ABB RAPID module: 9b54fd59.mod

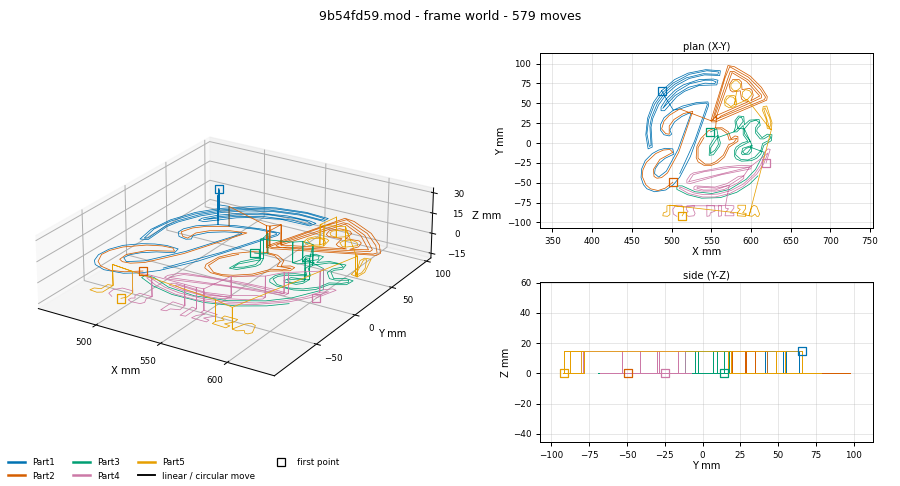
[picture p0: tool path of 9b54fd59.mod in frame world, 579 of 581 moves have a stored position in this frame; points joined in program order, loops and branches not executed]
MODULE ImageDraw
  ! Generated 2026-10-06 12:25 for ABB GoFa CRB 15000: 38 strokes
  PERS tooldata tPen:=[TRUE,[[0,0,120.0],[1,0,0,0]],[0.3,[0,0,60.0],[1,0,0,0],0,0,0]];
  PERS wobjdata wPaper:=[FALSE,TRUE,"",[[400,-110,0],[1,0,0,0]],[[0,0,0],[1,0,0,0]]];
  CONST robtarget pOrigin:=[[0,0,0],[0,1,0,0],[0,0,0,0],[9E9,9E9,9E9,9E9,9E9,9E9]];
  CONST jointtarget jHome:=[[0,0,0,0,30,0],[9E9,9E9,9E9,9E9,9E9,9E9]];
  CONST speeddata vDraw:=[40,100,5000,1000];
  CONST speeddata vApproach:=[20,100,5000,1000];
  CONST speeddata vTravel:=[200,200,5000,1000];

  PROC DrawImage()
    ConfL\Off;
    ConfJ\Off;
    MoveAbsJ jHome\NoEOffs,vTravel,fine,tPen;
    Part1;
    Part2;
    Part3;
    Part4;
    Part5;
    MoveAbsJ jHome\NoEOffs,vTravel,fine,tPen;
  ENDPROC

  PROC Part1()
    MoveL Offs(pOrigin,87.5,175.8,15.0),vTravel,z5,tPen\WObj:=wPaper;
    MoveL Offs(pOrigin,87.5,175.8,0.0),vApproach,fine,tPen\WObj:=wPaper;
    MoveL Offs(pOrigin,77.2,161.0,0.0),vDraw,z1,tPen\WObj:=wPaper;
    MoveL Offs(pOrigin,69.8,141.1,0.0),vDraw,z1,tPen\WObj:=wPaper;
    MoveL Offs(pOrigin,67.6,120.4,0.0),vDraw,z1,tPen\WObj:=wPaper;
    MoveL Offs(pOrigin,70.5,102.6,0.0),vDraw,z1,tPen\WObj:=wPaper;
    MoveL Offs(pOrigin,75.7,104.8,0.0),vDraw,z1,tPen\WObj:=wPaper;
    MoveL Offs(pOrigin,74.2,130.0,0.0),vDraw,z1,tPen\WObj:=wPaper;
    MoveL Offs(pOrigin,76.4,141.1,0.0),vDraw,z1,tPen\WObj:=wPaper;
    MoveL Offs(pOrigin,83.8,158.1,0.0),vDraw,z1,tPen\WObj:=wPaper;
    MoveL Offs(pOrigin,93.4,171.4,0.0),vDraw,z1,tPen\WObj:=wPaper;
    MoveL Offs(pOrigin,106.0,182.5,0.0),vDraw,z1,tPen\WObj:=wPaper;
    MoveL Offs(pOrigin,122.3,191.3,0.0),vDraw,z1,tPen\WObj:=wPaper;
    MoveL Offs(pOrigin,141.5,195.8,0.0),vDraw,z1,tPen\WObj:=wPaper;
    MoveL Offs(pOrigin,160.7,195.0,0.0),vDraw,z1,tPen\WObj:=wPaper;
    MoveL Offs(pOrigin,161.5,201.0,0.0),vDraw,z1,tPen\WObj:=wPaper;
    MoveL Offs(pOrigin,143.0,202.4,0.0),vDraw,z1,tPen\WObj:=wPaper;
    MoveL Offs(pOrigin,120.8,198.0,0.0),vDraw,z1,tPen\WObj:=wPaper;
    MoveL Offs(pOrigin,103.8,189.9,0.0),vDraw,z1,tPen\WObj:=wPaper;
    MoveL Offs(pOrigin,87.5,175.8,0.0),vDraw,fine,tPen\WObj:=wPaper;
    MoveL Offs(pOrigin,87.5,175.8,15.0),vApproach,z5,tPen\WObj:=wPaper;
    MoveL Offs(pOrigin,89.0,173.6,15.0),vTravel,z5,tPen\WObj:=wPaper;
    MoveL Offs(pOrigin,89.0,173.6,0.0),vApproach,fine,tPen\WObj:=wPaper;
    MoveL Offs(pOrigin,101.6,185.4,0.0),vDraw,z1,tPen\WObj:=wPaper;
    MoveL Offs(pOrigin,122.3,196.5,0.0),vDraw,z1,tPen\WObj:=wPaper;
    MoveL Offs(pOrigin,144.5,201.0,0.0),vDraw,z1,tPen\WObj:=wPaper;
    MoveL Offs(pOrigin,159.2,199.5,0.0),vDraw,z1,tPen\WObj:=wPaper;
    MoveL Offs(pOrigin,158.5,196.5,0.0),vDraw,z1,tPen\WObj:=wPaper;
    MoveL Offs(pOrigin,140.0,197.3,0.0),vDraw,z1,tPen\WObj:=wPaper;
    MoveL Offs(pOrigin,118.6,192.1,0.0),vDraw,z1,tPen\WObj:=wPaper;
    MoveL Offs(pOrigin,103.8,183.9,0.0),vDraw,z1,tPen\WObj:=wPaper;
    MoveL Offs(pOrigin,92.7,174.3,0.0),vDraw,z1,tPen\WObj:=wPaper;
    MoveL Offs(pOrigin,82.3,160.3,0.0),vDraw,z1,tPen\WObj:=wPaper;
    MoveL Offs(pOrigin,74.9,142.5,0.0),vDraw,z1,tPen\WObj:=wPaper;
    MoveL Offs(pOrigin,72.7,131.4,0.0),vDraw,z1,tPen\WObj:=wPaper;
    MoveL Offs(pOrigin,74.2,107.0,0.0),vDraw,z1,tPen\WObj:=wPaper;
    MoveL Offs(pOrigin,72.0,105.6,0.0),vDraw,z1,tPen\WObj:=wPaper;
    MoveL Offs(pOrigin,69.0,121.8,0.0),vDraw,z1,tPen\WObj:=wPaper;
    MoveL Offs(pOrigin,71.2,139.6,0.0),vDraw,z1,tPen\WObj:=wPaper;
    MoveL Offs(pOrigin,78.6,158.8,0.0),vDraw,z1,tPen\WObj:=wPaper;
    MoveL Offs(pOrigin,89.0,173.6,0.0),vDraw,fine,tPen\WObj:=wPaper;
    MoveL Offs(pOrigin,89.0,173.6,15.0),vApproach,z5,tPen\WObj:=wPaper;
    MoveL Offs(pOrigin,93.4,165.5,15.0),vTravel,z5,tPen\WObj:=wPaper;
    MoveL Offs(pOrigin,93.4,165.5,0.0),vApproach,fine,tPen\WObj:=wPaper;
    MoveL Offs(pOrigin,86.8,155.1,0.0),vDraw,z1,tPen\WObj:=wPaper;
    MoveL Offs(pOrigin,86.8,150.7,0.0),vDraw,z1,tPen\WObj:=wPaper;
    MoveL Offs(pOrigin,91.2,150.7,0.0),vDraw,z1,tPen\WObj:=wPaper;
    MoveL Offs(pOrigin,106.7,168.4,0.0),vDraw,z1,tPen\WObj:=wPaper;
    MoveL Offs(pOrigin,116.4,175.1,0.0),vDraw,z1,tPen\WObj:=wPaper;
    MoveL Offs(pOrigin,134.8,182.5,0.0),vDraw,z1,tPen\WObj:=wPaper;
    MoveL Offs(pOrigin,157.0,183.2,0.0),vDraw,z1,tPen\WObj:=wPaper;
    MoveL Offs(pOrigin,158.5,189.1,0.0),vDraw,z1,tPen\WObj:=wPaper;
    MoveL Offs(pOrigin,152.6,190.6,0.0),vDraw,z1,tPen\WObj:=wPaper;
    MoveL Offs(pOrigin,134.8,189.9,0.0),vDraw,z1,tPen\WObj:=wPaper;
    MoveL Offs(pOrigin,114.9,183.2,0.0),vDraw,z1,tPen\WObj:=wPaper;
    MoveL Offs(pOrigin,104.5,176.5,0.0),vDraw,z1,tPen\WObj:=wPaper;
    MoveL Offs(pOrigin,93.4,165.5,0.0),vDraw,fine,tPen\WObj:=wPaper;
    MoveL Offs(pOrigin,93.4,165.5,15.0),vApproach,z5,tPen\WObj:=wPaper;
    MoveL Offs(pOrigin,94.9,163.2,15.0),vTravel,z5,tPen\WObj:=wPaper;
    MoveL Offs(pOrigin,94.9,163.2,0.0),vApproach,fine,tPen\WObj:=wPaper;
    MoveL Offs(pOrigin,106.7,175.1,0.0),vDraw,z1,tPen\WObj:=wPaper;
    MoveL Offs(pOrigin,123.0,184.7,0.0),vDraw,z1,tPen\WObj:=wPaper;
    MoveL Offs(pOrigin,142.2,189.1,0.0),vDraw,z1,tPen\WObj:=wPaper;
    MoveL Offs(pOrigin,151.1,189.1,0.0),vDraw,z1,tPen\WObj:=wPaper;
    MoveL Offs(pOrigin,156.3,186.9,0.0),vDraw,z1,tPen\WObj:=wPaper;
    MoveL Offs(pOrigin,154.1,184.7,0.0),vDraw,z1,tPen\WObj:=wPaper;
    MoveL Offs(pOrigin,142.2,185.4,0.0),vDraw,z1,tPen\WObj:=wPaper;
    MoveL Offs(pOrigin,121.5,180.2,0.0),vDraw,z1,tPen\WObj:=wPaper;
    MoveL Offs(pOrigin,104.5,169.9,0.0),vDraw,z1,tPen\WObj:=wPaper;
    MoveL Offs(pOrigin,89.0,153.6,0.0),vDraw,z1,tPen\WObj:=wPaper;
    MoveL Offs(pOrigin,94.9,163.2,0.0),vDraw,fine,tPen\WObj:=wPaper;
    MoveL Offs(pOrigin,94.9,163.2,15.0),vApproach,z5,tPen\WObj:=wPaper;
    MoveL Offs(pOrigin,102.3,151.4,15.0),vTravel,z5,tPen\WObj:=wPaper;
    MoveL Offs(pOrigin,102.3,151.4,0.0),vApproach,fine,tPen\WObj:=wPaper;
    MoveL Offs(pOrigin,90.5,141.8,0.0),vDraw,z1,tPen\WObj:=wPaper;
    MoveL Offs(pOrigin,86.0,132.9,0.0),vDraw,z1,tPen\WObj:=wPaper;
    MoveL Offs(pOrigin,86.0,126.3,0.0),vDraw,z1,tPen\WObj:=wPaper;
    MoveL Offs(pOrigin,90.5,120.4,0.0),vDraw,z1,tPen\WObj:=wPaper;
    MoveL Offs(pOrigin,97.1,118.9,0.0),vDraw,z1,tPen\WObj:=wPaper;
    MoveL Offs(pOrigin,100.1,121.1,0.0),vDraw,z1,tPen\WObj:=wPaper;
    MoveL Offs(pOrigin,97.9,126.3,0.0),vDraw,z1,tPen\WObj:=wPaper;
    MoveL Offs(pOrigin,103.8,136.6,0.0),vDraw,z1,tPen\WObj:=wPaper;
    MoveL Offs(pOrigin,112.7,143.3,0.0),vDraw,z1,tPen\WObj:=wPaper;
    MoveL Offs(pOrigin,122.3,147.7,0.0),vDraw,z1,tPen\WObj:=wPaper;
    MoveL Offs(pOrigin,124.5,147.0,0.0),vDraw,z1,tPen\WObj:=wPaper;
    MoveL Offs(pOrigin,108.2,101.9,0.0),vDraw,z1,tPen\WObj:=wPaper;
    MoveL Offs(pOrigin,93.4,74.5,0.0),vDraw,z1,tPen\WObj:=wPaper;
    MoveL Offs(pOrigin,83.8,67.1,0.0),vDraw,z1,tPen\WObj:=wPaper;
    MoveL Offs(pOrigin,78.6,71.5,0.0),vDraw,z1,tPen\WObj:=wPaper;
    MoveL Offs(pOrigin,79.4,77.5,0.0),vDraw,z1,tPen\WObj:=wPaper;
    MoveL Offs(pOrigin,83.8,84.1,0.0),vDraw,z1,tPen\WObj:=wPaper;
    MoveL Offs(pOrigin,92.0,90.8,0.0),vDraw,z1,tPen\WObj:=wPaper;
    MoveL Offs(pOrigin,103.0,96.0,0.0),vDraw,z1,tPen\WObj:=wPaper;
    MoveL Offs(pOrigin,101.6,102.6,0.0),vDraw,z1,tPen\WObj:=wPaper;
    MoveL Offs(pOrigin,92.0,103.3,0.0),vDraw,z1,tPen\WObj:=wPaper;
    MoveL Offs(pOrigin,83.8,101.1,0.0),vDraw,z1,tPen\WObj:=wPaper;
    MoveL Offs(pOrigin,75.7,96.7,0.0),vDraw,z1,tPen\WObj:=wPaper;
    MoveL Offs(pOrigin,66.8,87.8,0.0),vDraw,z1,tPen\WObj:=wPaper;
    MoveL Offs(pOrigin,62.4,77.5,0.0),vDraw,z1,tPen\WObj:=wPaper;
    MoveL Offs(pOrigin,61.6,66.4,0.0),vDraw,z1,tPen\WObj:=wPaper;
    MoveL Offs(pOrigin,64.6,57.5,0.0),vDraw,z1,tPen\WObj:=wPaper;
    MoveL Offs(pOrigin,69.0,52.3,0.0),vDraw,z1,tPen\WObj:=wPaper;
    MoveL Offs(pOrigin,78.6,48.6,0.0),vDraw,z1,tPen\WObj:=wPaper;
    MoveL Offs(pOrigin,92.7,50.8,0.0),vDraw,z1,tPen\WObj:=wPaper;
    MoveL Offs(pOrigin,102.3,57.5,0.0),vDraw,z1,tPen\WObj:=wPaper;
    MoveL Offs(pOrigin,110.4,67.1,0.0),vDraw,z1,tPen\WObj:=wPaper;
    MoveL Offs(pOrigin,123.8,93.0,0.0),vDraw,z1,tPen\WObj:=wPaper;
    MoveL Offs(pOrigin,146.7,157.3,0.0),vDraw,z1,tPen\WObj:=wPaper;
    MoveL Offs(pOrigin,145.9,161.8,0.0),vDraw,z1,tPen\WObj:=wPaper;
    MoveL Offs(pOrigin,131.9,161.0,0.0),vDraw,z1,tPen\WObj:=wPaper;
    MoveL Offs(pOrigin,114.1,156.6,0.0),vDraw,z1,tPen\WObj:=wPaper;
    MoveL Offs(pOrigin,102.3,151.4,0.0),vDraw,fine,tPen\WObj:=wPaper;
    MoveL Offs(pOrigin,102.3,151.4,15.0),vApproach,z5,tPen\WObj:=wPaper;
    MoveL Offs(pOrigin,110.4,152.9,15.0),vTravel,z5,tPen\WObj:=wPaper;
    MoveL Offs(pOrigin,110.4,152.9,0.0),vApproach,fine,tPen\WObj:=wPaper;
    MoveL Offs(pOrigin,128.9,158.8,0.0),vDraw,z1,tPen\WObj:=wPaper;
    MoveL Offs(pOrigin,143.7,160.3,0.0),vDraw,z1,tPen\WObj:=wPaper;
    MoveL Offs(pOrigin,145.2,158.8,0.0),vDraw,z1,tPen\WObj:=wPaper;
    MoveL Offs(pOrigin,128.9,112.2,0.0),vDraw,z1,tPen\WObj:=wPaper;
    MoveL Offs(pOrigin,110.4,71.5,0.0),vDraw,z1,tPen\WObj:=wPaper;
  ENDPROC

  PROC Part2()
    MoveL Offs(pOrigin,101.6,60.5,0.0),vDraw,z1,tPen\WObj:=wPaper;
    MoveL Offs(pOrigin,92.0,53.1,0.0),vDraw,z1,tPen\WObj:=wPaper;
    MoveL Offs(pOrigin,83.1,50.1,0.0),vDraw,z1,tPen\WObj:=wPaper;
    MoveL Offs(pOrigin,73.5,52.3,0.0),vDraw,z1,tPen\WObj:=wPaper;
    MoveL Offs(pOrigin,67.6,57.5,0.0),vDraw,z1,tPen\WObj:=wPaper;
    MoveL Offs(pOrigin,63.1,67.9,0.0),vDraw,z1,tPen\WObj:=wPaper;
    MoveL Offs(pOrigin,63.9,76.0,0.0),vDraw,z1,tPen\WObj:=wPaper;
    MoveL Offs(pOrigin,68.3,85.6,0.0),vDraw,z1,tPen\WObj:=wPaper;
    MoveL Offs(pOrigin,80.1,96.7,0.0),vDraw,z1,tPen\WObj:=wPaper;
    MoveL Offs(pOrigin,89.7,101.1,0.0),vDraw,z1,tPen\WObj:=wPaper;
    MoveL Offs(pOrigin,97.9,101.9,0.0),vDraw,z1,tPen\WObj:=wPaper;
    MoveL Offs(pOrigin,101.6,98.2,0.0),vDraw,z1,tPen\WObj:=wPaper;
    MoveL Offs(pOrigin,85.3,89.3,0.0),vDraw,z1,tPen\WObj:=wPaper;
    MoveL Offs(pOrigin,77.2,76.7,0.0),vDraw,z1,tPen\WObj:=wPaper;
    MoveL Offs(pOrigin,77.9,67.9,0.0),vDraw,z1,tPen\WObj:=wPaper;
    MoveL Offs(pOrigin,81.6,65.6,0.0),vDraw,z1,tPen\WObj:=wPaper;
    MoveL Offs(pOrigin,87.5,66.4,0.0),vDraw,z1,tPen\WObj:=wPaper;
    MoveL Offs(pOrigin,94.9,72.3,0.0),vDraw,z1,tPen\WObj:=wPaper;
    MoveL Offs(pOrigin,109.0,98.2,0.0),vDraw,z1,tPen\WObj:=wPaper;
    MoveL Offs(pOrigin,126.7,149.9,0.0),vDraw,z1,tPen\WObj:=wPaper;
    MoveL Offs(pOrigin,114.9,147.0,0.0),vDraw,z1,tPen\WObj:=wPaper;
    MoveL Offs(pOrigin,103.0,139.6,0.0),vDraw,z1,tPen\WObj:=wPaper;
    MoveL Offs(pOrigin,97.1,131.4,0.0),vDraw,z1,tPen\WObj:=wPaper;
    MoveL Offs(pOrigin,97.1,121.1,0.0),vDraw,z1,tPen\WObj:=wPaper;
    MoveL Offs(pOrigin,92.7,121.8,0.0),vDraw,z1,tPen\WObj:=wPaper;
    MoveL Offs(pOrigin,87.5,127.7,0.0),vDraw,z1,tPen\WObj:=wPaper;
    MoveL Offs(pOrigin,90.5,137.4,0.0),vDraw,z1,tPen\WObj:=wPaper;
    MoveL Offs(pOrigin,97.1,144.8,0.0),vDraw,z1,tPen\WObj:=wPaper;
    MoveL Offs(pOrigin,110.4,152.9,0.0),vDraw,fine,tPen\WObj:=wPaper;
    MoveL Offs(pOrigin,110.4,152.9,15.0),vApproach,z5,tPen\WObj:=wPaper;
    MoveL Offs(pOrigin,149.6,138.1,15.0),vTravel,z5,tPen\WObj:=wPaper;
    MoveL Offs(pOrigin,149.6,138.1,0.0),vApproach,fine,tPen\WObj:=wPaper;
    MoveL Offs(pOrigin,150.4,136.6,0.0),vDraw,z1,tPen\WObj:=wPaper;
    MoveL Offs(pOrigin,155.5,136.6,0.0),vDraw,z1,tPen\WObj:=wPaper;
    MoveL Offs(pOrigin,219.9,164.0,0.0),vDraw,z1,tPen\WObj:=wPaper;
    MoveL Offs(pOrigin,220.6,168.4,0.0),vDraw,z1,tPen\WObj:=wPaper;
    MoveL Offs(pOrigin,213.2,180.2,0.0),vDraw,z1,tPen\WObj:=wPaper;
    MoveL Offs(pOrigin,199.2,194.3,0.0),vDraw,z1,tPen\WObj:=wPaper;
    MoveL Offs(pOrigin,179.2,206.1,0.0),vDraw,z1,tPen\WObj:=wPaper;
    MoveL Offs(pOrigin,171.1,207.6,0.0),vDraw,z1,tPen\WObj:=wPaper;
    MoveL Offs(pOrigin,149.6,138.1,0.0),vDraw,fine,tPen\WObj:=wPaper;
    MoveL Offs(pOrigin,149.6,138.1,15.0),vApproach,z5,tPen\WObj:=wPaper;
    MoveL Offs(pOrigin,151.8,138.8,15.0),vTravel,z5,tPen\WObj:=wPaper;
    MoveL Offs(pOrigin,151.8,138.8,0.0),vApproach,fine,tPen\WObj:=wPaper;
    MoveL Offs(pOrigin,167.4,192.1,0.0),vDraw,z1,tPen\WObj:=wPaper;
    MoveL Offs(pOrigin,173.3,206.1,0.0),vDraw,z1,tPen\WObj:=wPaper;
    MoveL Offs(pOrigin,197.0,192.8,0.0),vDraw,z1,tPen\WObj:=wPaper;
    MoveL Offs(pOrigin,211.7,178.0,0.0),vDraw,z1,tPen\WObj:=wPaper;
    MoveL Offs(pOrigin,218.4,167.7,0.0),vDraw,z1,tPen\WObj:=wPaper;
    MoveL Offs(pOrigin,216.9,164.7,0.0),vDraw,z1,tPen\WObj:=wPaper;
    MoveL Offs(pOrigin,159.2,141.1,0.0),vDraw,z1,tPen\WObj:=wPaper;
    MoveL Offs(pOrigin,162.2,144.0,0.0),vDraw,z1,tPen\WObj:=wPaper;
    MoveL Offs(pOrigin,213.2,166.9,0.0),vDraw,z1,tPen\WObj:=wPaper;
    MoveL Offs(pOrigin,213.2,170.6,0.0),vDraw,z1,tPen\WObj:=wPaper;
    MoveL Offs(pOrigin,197.0,189.1,0.0),vDraw,z1,tPen\WObj:=wPaper;
    MoveL Offs(pOrigin,178.5,200.2,0.0),vDraw,z1,tPen\WObj:=wPaper;
    MoveL Offs(pOrigin,174.0,200.2,0.0),vDraw,z1,tPen\WObj:=wPaper;
    MoveL Offs(pOrigin,154.8,144.8,0.0),vDraw,z1,tPen\WObj:=wPaper;
    MoveL Offs(pOrigin,154.8,141.8,0.0),vDraw,z1,tPen\WObj:=wPaper;
    MoveL Offs(pOrigin,159.2,141.1,0.0),vDraw,z1,tPen\WObj:=wPaper;
    MoveL Offs(pOrigin,154.1,138.1,0.0),vDraw,z1,tPen\WObj:=wPaper;
    MoveL Offs(pOrigin,151.8,138.8,0.0),vDraw,fine,tPen\WObj:=wPaper;
    MoveL Offs(pOrigin,151.8,138.8,15.0),vApproach,z5,tPen\WObj:=wPaper;
    MoveL Offs(pOrigin,157.0,144.8,15.0),vTravel,z5,tPen\WObj:=wPaper;
    MoveL Offs(pOrigin,157.0,144.8,0.0),vApproach,fine,tPen\WObj:=wPaper;
    MoveL Offs(pOrigin,176.2,198.7,0.0),vDraw,z1,tPen\WObj:=wPaper;
    MoveL Offs(pOrigin,194.7,187.6,0.0),vDraw,z1,tPen\WObj:=wPaper;
    MoveL Offs(pOrigin,211.0,169.2,0.0),vDraw,z1,tPen\WObj:=wPaper;
    MoveL Offs(pOrigin,199.9,163.2,0.0),vDraw,z1,tPen\WObj:=wPaper;
    MoveL Offs(pOrigin,202.9,169.9,0.0),vDraw,z1,tPen\WObj:=wPaper;
    MoveL Offs(pOrigin,201.4,176.5,0.0),vDraw,z1,tPen\WObj:=wPaper;
    MoveL Offs(pOrigin,198.4,178.8,0.0),vDraw,z1,tPen\WObj:=wPaper;
    MoveL Offs(pOrigin,188.8,177.3,0.0),vDraw,z1,tPen\WObj:=wPaper;
    MoveL Offs(pOrigin,188.1,186.9,0.0),vDraw,z1,tPen\WObj:=wPaper;
    MoveL Offs(pOrigin,185.1,189.9,0.0),vDraw,z1,tPen\WObj:=wPaper;
    MoveL Offs(pOrigin,177.0,189.9,0.0),vDraw,z1,tPen\WObj:=wPaper;
    MoveL Offs(pOrigin,172.6,183.2,0.0),vDraw,z1,tPen\WObj:=wPaper;
    MoveL Offs(pOrigin,174.0,176.5,0.0),vDraw,z1,tPen\WObj:=wPaper;
    MoveL Offs(pOrigin,177.0,174.3,0.0),vDraw,z1,tPen\WObj:=wPaper;
    MoveL Offs(pOrigin,186.6,175.8,0.0),vDraw,z1,tPen\WObj:=wPaper;
    MoveL Offs(pOrigin,188.1,165.5,0.0),vDraw,z1,tPen\WObj:=wPaper;
    MoveL Offs(pOrigin,191.0,163.2,0.0),vDraw,z1,tPen\WObj:=wPaper;
    MoveL Offs(pOrigin,197.7,162.5,0.0),vDraw,z1,tPen\WObj:=wPaper;
    MoveL Offs(pOrigin,157.0,144.8,0.0),vDraw,fine,tPen\WObj:=wPaper;
    MoveL Offs(pOrigin,157.0,144.8,15.0),vApproach,z5,tPen\WObj:=wPaper;
    MoveL Offs(pOrigin,155.5,129.2,15.0),vTravel,z5,tPen\WObj:=wPaper;
    MoveL Offs(pOrigin,155.5,129.2,0.0),vApproach,fine,tPen\WObj:=wPaper;
    MoveL Offs(pOrigin,146.7,125.5,0.0),vDraw,z1,tPen\WObj:=wPaper;
    MoveL Offs(pOrigin,137.1,115.9,0.0),vDraw,z1,tPen\WObj:=wPaper;
    MoveL Offs(pOrigin,131.9,105.6,0.0),vDraw,z1,tPen\WObj:=wPaper;
    MoveL Offs(pOrigin,131.1,91.5,0.0),vDraw,z1,tPen\WObj:=wPaper;
    MoveL Offs(pOrigin,133.4,86.3,0.0),vDraw,z1,tPen\WObj:=wPaper;
    MoveL Offs(pOrigin,140.8,81.9,0.0),vDraw,z1,tPen\WObj:=wPaper;
    MoveL Offs(pOrigin,150.4,81.9,0.0),vDraw,z1,tPen\WObj:=wPaper;
    MoveL Offs(pOrigin,157.8,84.9,0.0),vDraw,z1,tPen\WObj:=wPaper;
    MoveL Offs(pOrigin,166.6,92.3,0.0),vDraw,z1,tPen\WObj:=wPaper;
    MoveL Offs(pOrigin,172.6,104.8,0.0),vDraw,z1,tPen\WObj:=wPaper;
    MoveL Offs(pOrigin,183.6,112.2,0.0),vDraw,z1,tPen\WObj:=wPaper;
    MoveL Offs(pOrigin,183.6,118.1,0.0),vDraw,z1,tPen\WObj:=wPaper;
    MoveL Offs(pOrigin,179.9,118.9,0.0),vDraw,z1,tPen\WObj:=wPaper;
    MoveL Offs(pOrigin,174.8,115.2,0.0),vDraw,z1,tPen\WObj:=wPaper;
    MoveL Offs(pOrigin,171.8,124.0,0.0),vDraw,z1,tPen\WObj:=wPaper;
    MoveL Offs(pOrigin,163.7,129.2,0.0),vDraw,z1,tPen\WObj:=wPaper;
    MoveL Offs(pOrigin,155.5,129.2,0.0),vDraw,fine,tPen\WObj:=wPaper;
    MoveL Offs(pOrigin,155.5,129.2,15.0),vApproach,z5,tPen\WObj:=wPaper;
    MoveL Offs(pOrigin,157.0,127.7,15.0),vTravel,z5,tPen\WObj:=wPaper;
    MoveL Offs(pOrigin,157.0,127.7,0.0),vApproach,fine,tPen\WObj:=wPaper;
    MoveL Offs(pOrigin,162.2,127.7,0.0),vDraw,z1,tPen\WObj:=wPaper;
    MoveL Offs(pOrigin,170.3,121.8,0.0),vDraw,z1,tPen\WObj:=wPaper;
    MoveL Offs(pOrigin,172.6,113.7,0.0),vDraw,z1,tPen\WObj:=wPaper;
    MoveL Offs(pOrigin,182.2,115.9,0.0),vDraw,z1,tPen\WObj:=wPaper;
    MoveL Offs(pOrigin,178.5,110.7,0.0),vDraw,z1,tPen\WObj:=wPaper;
    MoveL Offs(pOrigin,171.8,107.8,0.0),vDraw,z1,tPen\WObj:=wPaper;
    MoveL Offs(pOrigin,165.2,94.5,0.0),vDraw,z1,tPen\WObj:=wPaper;
    MoveL Offs(pOrigin,155.5,86.3,0.0),vDraw,z1,tPen\WObj:=wPaper;
    MoveL Offs(pOrigin,148.9,83.4,0.0),vDraw,z1,tPen\WObj:=wPaper;
    MoveL Offs(pOrigin,142.2,83.4,0.0),vDraw,z1,tPen\WObj:=wPaper;
    MoveL Offs(pOrigin,133.4,90.8,0.0),vDraw,z1,tPen\WObj:=wPaper;
    MoveL Offs(pOrigin,133.4,104.1,0.0),vDraw,z1,tPen\WObj:=wPaper;
    MoveL Offs(pOrigin,140.8,116.7,0.0),vDraw,z1,tPen\WObj:=wPaper;
  ENDPROC

  PROC Part3()
    MoveL Offs(pOrigin,148.9,124.0,0.0),vDraw,z1,tPen\WObj:=wPaper;
    MoveL Offs(pOrigin,157.0,127.7,0.0),vDraw,fine,tPen\WObj:=wPaper;
    MoveL Offs(pOrigin,157.0,127.7,15.0),vApproach,z5,tPen\WObj:=wPaper;
    MoveL Offs(pOrigin,158.5,119.6,15.0),vTravel,z5,tPen\WObj:=wPaper;
    MoveL Offs(pOrigin,158.5,119.6,0.0),vApproach,fine,tPen\WObj:=wPaper;
    MoveL Offs(pOrigin,154.1,116.7,0.0),vDraw,z1,tPen\WObj:=wPaper;
    MoveL Offs(pOrigin,148.2,107.0,0.0),vDraw,z1,tPen\WObj:=wPaper;
    MoveL Offs(pOrigin,147.4,94.5,0.0),vDraw,z1,tPen\WObj:=wPaper;
    MoveL Offs(pOrigin,152.6,95.2,0.0),vDraw,z1,tPen\WObj:=wPaper;
    MoveL Offs(pOrigin,160.7,106.3,0.0),vDraw,z1,tPen\WObj:=wPaper;
    MoveL Offs(pOrigin,161.5,110.7,0.0),vDraw,z1,tPen\WObj:=wPaper;
    MoveL Offs(pOrigin,158.5,119.6,0.0),vDraw,fine,tPen\WObj:=wPaper;
    MoveL Offs(pOrigin,158.5,119.6,15.0),vApproach,z5,tPen\WObj:=wPaper;
    MoveL Offs(pOrigin,157.8,116.7,15.0),vTravel,z5,tPen\WObj:=wPaper;
    MoveL Offs(pOrigin,157.8,116.7,0.0),vApproach,fine,tPen\WObj:=wPaper;
    MoveL Offs(pOrigin,159.2,108.5,0.0),vDraw,z1,tPen\WObj:=wPaper;
    MoveL Offs(pOrigin,154.8,101.1,0.0),vDraw,z1,tPen\WObj:=wPaper;
    MoveL Offs(pOrigin,148.9,96.7,0.0),vDraw,z1,tPen\WObj:=wPaper;
    MoveL Offs(pOrigin,148.9,103.3,0.0),vDraw,z1,tPen\WObj:=wPaper;
    MoveL Offs(pOrigin,157.8,116.7,0.0),vDraw,fine,tPen\WObj:=wPaper;
    MoveL Offs(pOrigin,157.8,116.7,15.0),vApproach,z5,tPen\WObj:=wPaper;
    MoveL Offs(pOrigin,178.5,124.0,15.0),vTravel,z5,tPen\WObj:=wPaper;
    MoveL Offs(pOrigin,178.5,124.0,0.0),vApproach,fine,tPen\WObj:=wPaper;
    MoveL Offs(pOrigin,182.2,124.0,0.0),vDraw,z1,tPen\WObj:=wPaper;
    MoveL Offs(pOrigin,190.3,132.2,0.0),vDraw,z1,tPen\WObj:=wPaper;
    MoveL Offs(pOrigin,190.3,120.4,0.0),vDraw,z1,tPen\WObj:=wPaper;
    MoveL Offs(pOrigin,196.2,112.2,0.0),vDraw,z1,tPen\WObj:=wPaper;
    MoveL Offs(pOrigin,188.8,110.0,0.0),vDraw,z1,tPen\WObj:=wPaper;
    MoveL Offs(pOrigin,181.4,104.8,0.0),vDraw,z1,tPen\WObj:=wPaper;
    MoveL Offs(pOrigin,179.2,100.4,0.0),vDraw,z1,tPen\WObj:=wPaper;
    MoveL Offs(pOrigin,179.2,93.7,0.0),vDraw,z1,tPen\WObj:=wPaper;
    MoveL Offs(pOrigin,181.4,90.0,0.0),vDraw,z1,tPen\WObj:=wPaper;
    MoveL Offs(pOrigin,188.1,87.1,0.0),vDraw,z1,tPen\WObj:=wPaper;
    MoveL Offs(pOrigin,200.7,87.8,0.0),vDraw,z1,tPen\WObj:=wPaper;
    MoveL Offs(pOrigin,207.3,90.8,0.0),vDraw,z1,tPen\WObj:=wPaper;
    MoveL Offs(pOrigin,212.5,96.0,0.0),vDraw,z1,tPen\WObj:=wPaper;
    MoveL Offs(pOrigin,216.2,107.0,0.0),vDraw,z1,tPen\WObj:=wPaper;
    MoveL Offs(pOrigin,225.8,113.0,0.0),vDraw,z1,tPen\WObj:=wPaper;
    MoveL Offs(pOrigin,226.5,120.4,0.0),vDraw,z1,tPen\WObj:=wPaper;
    MoveL Offs(pOrigin,220.6,121.1,0.0),vDraw,z1,tPen\WObj:=wPaper;
    MoveL Offs(pOrigin,214.0,116.7,0.0),vDraw,z1,tPen\WObj:=wPaper;
    MoveL Offs(pOrigin,207.3,124.8,0.0),vDraw,z1,tPen\WObj:=wPaper;
    MoveL Offs(pOrigin,208.0,128.5,0.0),vDraw,z1,tPen\WObj:=wPaper;
    MoveL Offs(pOrigin,211.7,132.2,0.0),vDraw,z1,tPen\WObj:=wPaper;
    MoveL Offs(pOrigin,210.3,139.6,0.0),vDraw,z1,tPen\WObj:=wPaper;
    MoveL Offs(pOrigin,198.4,138.8,0.0),vDraw,z1,tPen\WObj:=wPaper;
    MoveL Offs(pOrigin,191.8,132.9,0.0),vDraw,z1,tPen\WObj:=wPaper;
    MoveL Offs(pOrigin,191.0,143.3,0.0),vDraw,z1,tPen\WObj:=wPaper;
    MoveL Offs(pOrigin,184.4,144.0,0.0),vDraw,z1,tPen\WObj:=wPaper;
    MoveL Offs(pOrigin,179.9,138.1,0.0),vDraw,z1,tPen\WObj:=wPaper;
    MoveL Offs(pOrigin,180.7,130.7,0.0),vDraw,z1,tPen\WObj:=wPaper;
    MoveL Offs(pOrigin,178.5,124.0,0.0),vDraw,fine,tPen\WObj:=wPaper;
    MoveL Offs(pOrigin,178.5,124.0,15.0),vApproach,z5,tPen\WObj:=wPaper;
    MoveL Offs(pOrigin,183.6,128.5,15.0),vTravel,z5,tPen\WObj:=wPaper;
    MoveL Offs(pOrigin,183.6,128.5,0.0),vApproach,fine,tPen\WObj:=wPaper;
    MoveL Offs(pOrigin,181.4,136.6,0.0),vDraw,z1,tPen\WObj:=wPaper;
    MoveL Offs(pOrigin,185.1,141.8,0.0),vDraw,z1,tPen\WObj:=wPaper;
    MoveL Offs(pOrigin,188.1,142.5,0.0),vDraw,z1,tPen\WObj:=wPaper;
    MoveL Offs(pOrigin,190.3,137.4,0.0),vDraw,z1,tPen\WObj:=wPaper;
    MoveL Offs(pOrigin,183.6,128.5,0.0),vDraw,fine,tPen\WObj:=wPaper;
    MoveL Offs(pOrigin,183.6,128.5,15.0),vApproach,z5,tPen\WObj:=wPaper;
    MoveL Offs(pOrigin,191.8,127.7,15.0),vTravel,z5,tPen\WObj:=wPaper;
    MoveL Offs(pOrigin,191.8,127.7,0.0),vApproach,fine,tPen\WObj:=wPaper;
    MoveL Offs(pOrigin,199.2,136.6,0.0),vDraw,z1,tPen\WObj:=wPaper;
    MoveL Offs(pOrigin,206.6,138.8,0.0),vDraw,z1,tPen\WObj:=wPaper;
    MoveL Offs(pOrigin,210.3,135.9,0.0),vDraw,z1,tPen\WObj:=wPaper;
    MoveL Offs(pOrigin,205.8,129.2,0.0),vDraw,z1,tPen\WObj:=wPaper;
    MoveL Offs(pOrigin,205.8,122.6,0.0),vDraw,z1,tPen\WObj:=wPaper;
    MoveL Offs(pOrigin,211.7,115.2,0.0),vDraw,z1,tPen\WObj:=wPaper;
    MoveL Offs(pOrigin,216.2,115.2,0.0),vDraw,z1,tPen\WObj:=wPaper;
    MoveL Offs(pOrigin,223.6,119.6,0.0),vDraw,z1,tPen\WObj:=wPaper;
    MoveL Offs(pOrigin,225.1,116.7,0.0),vDraw,z1,tPen\WObj:=wPaper;
    MoveL Offs(pOrigin,222.1,113.0,0.0),vDraw,z1,tPen\WObj:=wPaper;
    MoveL Offs(pOrigin,214.7,109.3,0.0),vDraw,z1,tPen\WObj:=wPaper;
    MoveL Offs(pOrigin,212.5,100.4,0.0),vDraw,z1,tPen\WObj:=wPaper;
    MoveL Offs(pOrigin,205.1,92.3,0.0),vDraw,z1,tPen\WObj:=wPaper;
    MoveL Offs(pOrigin,196.2,88.6,0.0),vDraw,z1,tPen\WObj:=wPaper;
    MoveL Offs(pOrigin,187.3,89.3,0.0),vDraw,z1,tPen\WObj:=wPaper;
    MoveL Offs(pOrigin,180.7,95.2,0.0),vDraw,z1,tPen\WObj:=wPaper;
    MoveL Offs(pOrigin,181.4,100.4,0.0),vDraw,z1,tPen\WObj:=wPaper;
    MoveL Offs(pOrigin,185.1,104.8,0.0),vDraw,z1,tPen\WObj:=wPaper;
    MoveL Offs(pOrigin,199.2,112.2,0.0),vDraw,z1,tPen\WObj:=wPaper;
    MoveL Offs(pOrigin,191.8,121.8,0.0),vDraw,z1,tPen\WObj:=wPaper;
    MoveL Offs(pOrigin,191.8,127.7,0.0),vDraw,fine,tPen\WObj:=wPaper;
    MoveL Offs(pOrigin,191.8,127.7,15.0),vApproach,z5,tPen\WObj:=wPaper;
    MoveL Offs(pOrigin,201.4,107.0,15.0),vTravel,z5,tPen\WObj:=wPaper;
    MoveL Offs(pOrigin,201.4,107.0,0.0),vApproach,fine,tPen\WObj:=wPaper;
    MoveL Offs(pOrigin,189.6,103.3,0.0),vDraw,z1,tPen\WObj:=wPaper;
    MoveL Offs(pOrigin,188.1,96.7,0.0),vDraw,z1,tPen\WObj:=wPaper;
    MoveL Offs(pOrigin,189.6,95.2,0.0),vDraw,z1,tPen\WObj:=wPaper;
    MoveL Offs(pOrigin,197.7,96.0,0.0),vDraw,z1,tPen\WObj:=wPaper;
    MoveL Offs(pOrigin,200.7,99.6,0.0),vDraw,z1,tPen\WObj:=wPaper;
    MoveL Offs(pOrigin,201.4,107.0,0.0),vDraw,fine,tPen\WObj:=wPaper;
    MoveL Offs(pOrigin,201.4,107.0,15.0),vApproach,z5,tPen\WObj:=wPaper;
    MoveL Offs(pOrigin,199.2,104.8,15.0),vTravel,z5,tPen\WObj:=wPaper;
    MoveL Offs(pOrigin,199.2,104.8,0.0),vApproach,fine,tPen\WObj:=wPaper;
    MoveL Offs(pOrigin,199.9,103.3,0.0),vDraw,z1,tPen\WObj:=wPaper;
    MoveL Offs(pOrigin,195.5,97.4,0.0),vDraw,z1,tPen\WObj:=wPaper;
    MoveL Offs(pOrigin,191.8,96.7,0.0),vDraw,z1,tPen\WObj:=wPaper;
    MoveL Offs(pOrigin,189.6,98.9,0.0),vDraw,z1,tPen\WObj:=wPaper;
    MoveL Offs(pOrigin,194.0,103.3,0.0),vDraw,z1,tPen\WObj:=wPaper;
    MoveL Offs(pOrigin,199.2,104.8,0.0),vDraw,fine,tPen\WObj:=wPaper;
    MoveL Offs(pOrigin,199.2,104.8,15.0),vApproach,z5,tPen\WObj:=wPaper;
    MoveL Offs(pOrigin,216.9,98.2,15.0),vTravel,z5,tPen\WObj:=wPaper;
    MoveL Offs(pOrigin,216.9,98.2,0.0),vApproach,fine,tPen\WObj:=wPaper;
    MoveL Offs(pOrigin,205.8,76.7,0.0),vDraw,z1,tPen\WObj:=wPaper;
    MoveL Offs(pOrigin,194.0,64.2,0.0),vDraw,z1,tPen\WObj:=wPaper;
    MoveL Offs(pOrigin,173.3,51.6,0.0),vDraw,z1,tPen\WObj:=wPaper;
    MoveL Offs(pOrigin,151.1,46.4,0.0),vDraw,z1,tPen\WObj:=wPaper;
    MoveL Offs(pOrigin,129.7,48.6,0.0),vDraw,z1,tPen\WObj:=wPaper;
    MoveL Offs(pOrigin,113.4,56.0,0.0),vDraw,z1,tPen\WObj:=wPaper;
    MoveL Offs(pOrigin,109.0,56.0,0.0),vDraw,z1,tPen\WObj:=wPaper;
    MoveL Offs(pOrigin,106.7,54.5,0.0),vDraw,z1,tPen\WObj:=wPaper;
    MoveL Offs(pOrigin,106.7,51.6,0.0),vDraw,z1,tPen\WObj:=wPaper;
    MoveL Offs(pOrigin,120.1,44.9,0.0),vDraw,z1,tPen\WObj:=wPaper;
    MoveL Offs(pOrigin,137.8,40.5,0.0),vDraw,z1,tPen\WObj:=wPaper;
    MoveL Offs(pOrigin,161.5,41.2,0.0),vDraw,z1,tPen\WObj:=wPaper;
    MoveL Offs(pOrigin,182.2,47.9,0.0),vDraw,z1,tPen\WObj:=wPaper;
    MoveL Offs(pOrigin,198.4,58.2,0.0),vDraw,z1,tPen\WObj:=wPaper;
    MoveL Offs(pOrigin,208.8,68.6,0.0),vDraw,z1,tPen\WObj:=wPaper;
  ENDPROC

  PROC Part4()
    MoveL Offs(pOrigin,219.1,84.9,0.0),vDraw,z1,tPen\WObj:=wPaper;
    MoveL Offs(pOrigin,224.3,101.9,0.0),vDraw,z1,tPen\WObj:=wPaper;
    MoveL Offs(pOrigin,221.4,102.6,0.0),vDraw,z1,tPen\WObj:=wPaper;
    MoveL Offs(pOrigin,216.9,98.2,0.0),vDraw,fine,tPen\WObj:=wPaper;
    MoveL Offs(pOrigin,216.9,98.2,15.0),vApproach,z5,tPen\WObj:=wPaper;
    MoveL Offs(pOrigin,216.9,93.7,15.0),vTravel,z5,tPen\WObj:=wPaper;
    MoveL Offs(pOrigin,216.9,93.7,0.0),vApproach,fine,tPen\WObj:=wPaper;
    MoveL Offs(pOrigin,221.4,97.4,0.0),vDraw,z1,tPen\WObj:=wPaper;
    MoveL Offs(pOrigin,216.2,84.1,0.0),vDraw,z1,tPen\WObj:=wPaper;
    MoveL Offs(pOrigin,207.3,70.8,0.0),vDraw,z1,tPen\WObj:=wPaper;
    MoveL Offs(pOrigin,190.3,55.3,0.0),vDraw,z1,tPen\WObj:=wPaper;
    MoveL Offs(pOrigin,173.3,46.4,0.0),vDraw,z1,tPen\WObj:=wPaper;
    MoveL Offs(pOrigin,154.8,42.0,0.0),vDraw,z1,tPen\WObj:=wPaper;
    MoveL Offs(pOrigin,139.3,42.0,0.0),vDraw,z1,tPen\WObj:=wPaper;
    MoveL Offs(pOrigin,121.5,46.4,0.0),vDraw,z1,tPen\WObj:=wPaper;
    MoveL Offs(pOrigin,109.7,53.1,0.0),vDraw,z1,tPen\WObj:=wPaper;
    MoveL Offs(pOrigin,111.2,54.5,0.0),vDraw,z1,tPen\WObj:=wPaper;
    MoveL Offs(pOrigin,128.2,47.1,0.0),vDraw,z1,tPen\WObj:=wPaper;
    MoveL Offs(pOrigin,140.8,44.9,0.0),vDraw,z1,tPen\WObj:=wPaper;
    MoveL Offs(pOrigin,158.5,45.7,0.0),vDraw,z1,tPen\WObj:=wPaper;
    MoveL Offs(pOrigin,174.8,50.1,0.0),vDraw,z1,tPen\WObj:=wPaper;
    MoveL Offs(pOrigin,190.3,58.2,0.0),vDraw,z1,tPen\WObj:=wPaper;
    MoveL Offs(pOrigin,204.3,70.8,0.0),vDraw,z1,tPen\WObj:=wPaper;
    MoveL Offs(pOrigin,212.5,82.6,0.0),vDraw,z1,tPen\WObj:=wPaper;
    MoveL Offs(pOrigin,216.9,93.7,0.0),vDraw,fine,tPen\WObj:=wPaper;
    MoveL Offs(pOrigin,216.9,93.7,15.0),vApproach,z5,tPen\WObj:=wPaper;
    MoveL Offs(pOrigin,200.7,81.2,15.0),vTravel,z5,tPen\WObj:=wPaper;
    MoveL Offs(pOrigin,200.7,81.2,0.0),vApproach,fine,tPen\WObj:=wPaper;
    MoveL Offs(pOrigin,188.1,81.9,0.0),vDraw,z1,tPen\WObj:=wPaper;
    MoveL Offs(pOrigin,165.2,79.7,0.0),vDraw,z1,tPen\WObj:=wPaper;
    MoveL Offs(pOrigin,127.4,72.3,0.0),vDraw,z1,tPen\WObj:=wPaper;
    MoveL Offs(pOrigin,123.8,70.1,0.0),vDraw,z1,tPen\WObj:=wPaper;
    MoveL Offs(pOrigin,119.3,63.4,0.0),vDraw,z1,tPen\WObj:=wPaper;
    MoveL Offs(pOrigin,119.3,59.7,0.0),vDraw,z1,tPen\WObj:=wPaper;
    MoveL Offs(pOrigin,123.8,59.0,0.0),vDraw,z1,tPen\WObj:=wPaper;
    MoveL Offs(pOrigin,162.9,70.1,0.0),vDraw,z1,tPen\WObj:=wPaper;
    MoveL Offs(pOrigin,199.9,77.5,0.0),vDraw,z1,tPen\WObj:=wPaper;
    MoveL Offs(pOrigin,200.7,81.2,0.0),vDraw,fine,tPen\WObj:=wPaper;
    MoveL Offs(pOrigin,200.7,81.2,15.0),vApproach,z5,tPen\WObj:=wPaper;
    MoveL Offs(pOrigin,198.4,79.7,15.0),vTravel,z5,tPen\WObj:=wPaper;
    MoveL Offs(pOrigin,198.4,79.7,0.0),vApproach,fine,tPen\WObj:=wPaper;
    MoveL Offs(pOrigin,121.5,61.2,0.0),vDraw,z1,tPen\WObj:=wPaper;
    MoveL Offs(pOrigin,127.4,70.1,0.0),vDraw,z1,tPen\WObj:=wPaper;
    MoveL Offs(pOrigin,140.8,73.8,0.0),vDraw,z1,tPen\WObj:=wPaper;
    MoveL Offs(pOrigin,173.3,78.9,0.0),vDraw,z1,tPen\WObj:=wPaper;
    MoveL Offs(pOrigin,198.4,79.7,0.0),vDraw,fine,tPen\WObj:=wPaper;
    MoveL Offs(pOrigin,198.4,79.7,15.0),vApproach,z5,tPen\WObj:=wPaper;
    MoveL Offs(pOrigin,191.0,68.6,15.0),vTravel,z5,tPen\WObj:=wPaper;
    MoveL Offs(pOrigin,191.0,68.6,0.0),vApproach,fine,tPen\WObj:=wPaper;
    MoveL Offs(pOrigin,184.4,67.9,0.0),vDraw,z1,tPen\WObj:=wPaper;
    MoveL Offs(pOrigin,170.3,59.0,0.0),vDraw,z1,tPen\WObj:=wPaper;
    MoveL Offs(pOrigin,154.8,54.5,0.0),vDraw,z1,tPen\WObj:=wPaper;
    MoveL Offs(pOrigin,130.4,56.0,0.0),vDraw,z1,tPen\WObj:=wPaper;
    MoveL Offs(pOrigin,128.2,54.5,0.0),vDraw,z1,tPen\WObj:=wPaper;
    MoveL Offs(pOrigin,128.2,51.6,0.0),vDraw,z1,tPen\WObj:=wPaper;
    MoveL Offs(pOrigin,138.5,49.4,0.0),vDraw,z1,tPen\WObj:=wPaper;
    MoveL Offs(pOrigin,156.3,49.4,0.0),vDraw,z1,tPen\WObj:=wPaper;
    MoveL Offs(pOrigin,166.6,51.6,0.0),vDraw,z1,tPen\WObj:=wPaper;
    MoveL Offs(pOrigin,183.6,59.7,0.0),vDraw,z1,tPen\WObj:=wPaper;
    MoveL Offs(pOrigin,191.0,65.6,0.0),vDraw,z1,tPen\WObj:=wPaper;
    MoveL Offs(pOrigin,191.0,68.6,0.0),vDraw,fine,tPen\WObj:=wPaper;
    MoveL Offs(pOrigin,191.0,68.6,15.0),vApproach,z5,tPen\WObj:=wPaper;
    MoveL Offs(pOrigin,172.6,56.8,15.0),vTravel,z5,tPen\WObj:=wPaper;
    MoveL Offs(pOrigin,172.6,56.8,0.0),vApproach,fine,tPen\WObj:=wPaper;
    MoveL Offs(pOrigin,154.8,50.8,0.0),vDraw,z1,tPen\WObj:=wPaper;
    MoveL Offs(pOrigin,140.0,50.8,0.0),vDraw,z1,tPen\WObj:=wPaper;
    MoveL Offs(pOrigin,131.9,53.1,0.0),vDraw,z1,tPen\WObj:=wPaper;
    MoveL Offs(pOrigin,132.6,54.5,0.0),vDraw,z1,tPen\WObj:=wPaper;
    MoveL Offs(pOrigin,156.3,53.1,0.0),vDraw,z1,tPen\WObj:=wPaper;
    MoveL Offs(pOrigin,172.6,56.8,0.0),vDraw,fine,tPen\WObj:=wPaper;
    MoveL Offs(pOrigin,172.6,56.8,15.0),vApproach,z5,tPen\WObj:=wPaper;
    MoveL Offs(pOrigin,168.1,31.6,15.0),vTravel,z5,tPen\WObj:=wPaper;
    MoveL Offs(pOrigin,168.1,31.6,0.0),vApproach,fine,tPen\WObj:=wPaper;
    MoveL Offs(pOrigin,168.1,27.9,0.0),vDraw,z1,tPen\WObj:=wPaper;
    MoveL Offs(pOrigin,171.8,27.2,0.0),vDraw,z1,tPen\WObj:=wPaper;
    MoveL Offs(pOrigin,168.1,22.7,0.0),vDraw,z1,tPen\WObj:=wPaper;
    MoveL Offs(pOrigin,167.4,18.3,0.0),vDraw,z1,tPen\WObj:=wPaper;
    MoveL Offs(pOrigin,178.5,18.3,0.0),vDraw,z1,tPen\WObj:=wPaper;
    MoveL Offs(pOrigin,178.5,21.3,0.0),vDraw,z1,tPen\WObj:=wPaper;
    MoveL Offs(pOrigin,174.0,22.0,0.0),vDraw,z1,tPen\WObj:=wPaper;
    MoveL Offs(pOrigin,178.5,27.9,0.0),vDraw,z1,tPen\WObj:=wPaper;
    MoveL Offs(pOrigin,178.5,30.9,0.0),vDraw,z1,tPen\WObj:=wPaper;
    MoveL Offs(pOrigin,168.1,31.6,0.0),vDraw,fine,tPen\WObj:=wPaper;
    MoveL Offs(pOrigin,168.1,31.6,15.0),vApproach,z5,tPen\WObj:=wPaper;
    MoveL Offs(pOrigin,162.9,30.9,15.0),vTravel,z5,tPen\WObj:=wPaper;
    MoveL Offs(pOrigin,162.9,30.9,0.0),vApproach,fine,tPen\WObj:=wPaper;
    MoveL Offs(pOrigin,159.2,31.6,0.0),vDraw,z1,tPen\WObj:=wPaper;
    MoveL Offs(pOrigin,159.2,17.6,0.0),vDraw,z1,tPen\WObj:=wPaper;
    MoveL Offs(pOrigin,162.9,18.3,0.0),vDraw,z1,tPen\WObj:=wPaper;
    MoveL Offs(pOrigin,162.9,30.9,0.0),vDraw,fine,tPen\WObj:=wPaper;
    MoveL Offs(pOrigin,162.9,30.9,15.0),vApproach,z5,tPen\WObj:=wPaper;
    MoveL Offs(pOrigin,154.1,30.9,15.0),vTravel,z5,tPen\WObj:=wPaper;
    MoveL Offs(pOrigin,154.1,30.9,0.0),vApproach,fine,tPen\WObj:=wPaper;
    MoveL Offs(pOrigin,144.5,31.6,0.0),vDraw,z1,tPen\WObj:=wPaper;
    MoveL Offs(pOrigin,144.5,17.6,0.0),vDraw,z1,tPen\WObj:=wPaper;
    MoveL Offs(pOrigin,148.2,18.3,0.0),vDraw,z1,tPen\WObj:=wPaper;
    MoveL Offs(pOrigin,148.9,22.0,0.0),vDraw,z1,tPen\WObj:=wPaper;
    MoveL Offs(pOrigin,154.8,24.2,0.0),vDraw,z1,tPen\WObj:=wPaper;
    MoveL Offs(pOrigin,154.1,30.9,0.0),vDraw,fine,tPen\WObj:=wPaper;
    MoveL Offs(pOrigin,154.1,30.9,15.0),vApproach,z5,tPen\WObj:=wPaper;
    MoveL Offs(pOrigin,128.9,30.9,15.0),vTravel,z5,tPen\WObj:=wPaper;
    MoveL Offs(pOrigin,128.9,30.9,0.0),vApproach,fine,tPen\WObj:=wPaper;
    MoveL Offs(pOrigin,119.3,30.9,0.0),vDraw,z1,tPen\WObj:=wPaper;
    MoveL Offs(pOrigin,118.6,26.4,0.0),vDraw,z1,tPen\WObj:=wPaper;
    MoveL Offs(pOrigin,120.8,23.5,0.0),vDraw,z1,tPen\WObj:=wPaper;
    MoveL Offs(pOrigin,118.6,22.0,0.0),vDraw,z1,tPen\WObj:=wPaper;
    MoveL Offs(pOrigin,118.6,19.0,0.0),vDraw,z1,tPen\WObj:=wPaper;
    MoveL Offs(pOrigin,121.5,17.6,0.0),vDraw,z1,tPen\WObj:=wPaper;
    MoveL Offs(pOrigin,128.2,18.3,0.0),vDraw,z1,tPen\WObj:=wPaper;
    MoveL Offs(pOrigin,129.7,21.3,0.0),vDraw,z1,tPen\WObj:=wPaper;
    MoveL Offs(pOrigin,127.4,26.4,0.0),vDraw,z1,tPen\WObj:=wPaper;
    MoveL Offs(pOrigin,128.9,30.9,0.0),vDraw,fine,tPen\WObj:=wPaper;
    MoveL Offs(pOrigin,128.9,30.9,15.0),vApproach,z5,tPen\WObj:=wPaper;
    MoveL Offs(pOrigin,114.9,29.4,15.0),vTravel,z5,tPen\WObj:=wPaper;
    MoveL Offs(pOrigin,114.9,29.4,0.0),vApproach,fine,tPen\WObj:=wPaper;
    MoveL Offs(pOrigin,112.7,31.6,0.0),vDraw,z1,tPen\WObj:=wPaper;
    MoveL Offs(pOrigin,105.3,31.6,0.0),vDraw,z1,tPen\WObj:=wPaper;
    MoveL Offs(pOrigin,101.6,26.4,0.0),vDraw,z1,tPen\WObj:=wPaper;
    MoveL Offs(pOrigin,102.3,20.5,0.0),vDraw,z1,tPen\WObj:=wPaper;
    MoveL Offs(pOrigin,106.7,17.6,0.0),vDraw,z1,tPen\WObj:=wPaper;
  ENDPROC

  PROC Part5()
    MoveL Offs(pOrigin,113.4,18.3,0.0),vDraw,z1,tPen\WObj:=wPaper;
    MoveL Offs(pOrigin,115.6,22.0,0.0),vDraw,z1,tPen\WObj:=wPaper;
    MoveL Offs(pOrigin,114.9,29.4,0.0),vDraw,fine,tPen\WObj:=wPaper;
    MoveL Offs(pOrigin,114.9,29.4,15.0),vApproach,z5,tPen\WObj:=wPaper;
    MoveL Offs(pOrigin,97.9,31.6,15.0),vTravel,z5,tPen\WObj:=wPaper;
    MoveL Offs(pOrigin,97.9,31.6,0.0),vApproach,fine,tPen\WObj:=wPaper;
    MoveL Offs(pOrigin,94.2,30.9,0.0),vDraw,z1,tPen\WObj:=wPaper;
    MoveL Offs(pOrigin,94.2,23.5,0.0),vDraw,z1,tPen\WObj:=wPaper;
    MoveL Offs(pOrigin,89.7,22.0,0.0),vDraw,z1,tPen\WObj:=wPaper;
    MoveL Offs(pOrigin,89.0,18.3,0.0),vDraw,z1,tPen\WObj:=wPaper;
    MoveL Offs(pOrigin,94.9,17.6,0.0),vDraw,z1,tPen\WObj:=wPaper;
    MoveL Offs(pOrigin,97.9,19.8,0.0),vDraw,z1,tPen\WObj:=wPaper;
    MoveL Offs(pOrigin,97.9,31.6,0.0),vDraw,fine,tPen\WObj:=wPaper;
    MoveL Offs(pOrigin,97.9,31.6,15.0),vApproach,z5,tPen\WObj:=wPaper;
    MoveL Offs(pOrigin,182.9,22.0,15.0),vTravel,z5,tPen\WObj:=wPaper;
    MoveL Offs(pOrigin,182.9,22.0,0.0),vApproach,fine,tPen\WObj:=wPaper;
    MoveL Offs(pOrigin,182.9,18.3,0.0),vDraw,z1,tPen\WObj:=wPaper;
    MoveL Offs(pOrigin,193.3,17.6,0.0),vDraw,z1,tPen\WObj:=wPaper;
    MoveL Offs(pOrigin,194.0,21.3,0.0),vDraw,z1,tPen\WObj:=wPaper;
    MoveL Offs(pOrigin,189.6,22.0,0.0),vDraw,z1,tPen\WObj:=wPaper;
    MoveL Offs(pOrigin,193.3,27.2,0.0),vDraw,z1,tPen\WObj:=wPaper;
    MoveL Offs(pOrigin,193.3,31.6,0.0),vDraw,z1,tPen\WObj:=wPaper;
    MoveL Offs(pOrigin,183.6,31.6,0.0),vDraw,z1,tPen\WObj:=wPaper;
    MoveL Offs(pOrigin,183.6,27.9,0.0),vDraw,z1,tPen\WObj:=wPaper;
    MoveL Offs(pOrigin,186.6,26.4,0.0),vDraw,z1,tPen\WObj:=wPaper;
    MoveL Offs(pOrigin,182.9,22.0,0.0),vDraw,fine,tPen\WObj:=wPaper;
    MoveL Offs(pOrigin,182.9,22.0,15.0),vApproach,z5,tPen\WObj:=wPaper;
    MoveL Offs(pOrigin,197.7,18.3,15.0),vTravel,z5,tPen\WObj:=wPaper;
    MoveL Offs(pOrigin,197.7,18.3,0.0),vApproach,fine,tPen\WObj:=wPaper;
    MoveL Offs(pOrigin,201.4,17.6,0.0),vDraw,z1,tPen\WObj:=wPaper;
    MoveL Offs(pOrigin,205.1,20.5,0.0),vDraw,z1,tPen\WObj:=wPaper;
    MoveL Offs(pOrigin,207.3,17.6,0.0),vDraw,z1,tPen\WObj:=wPaper;
    MoveL Offs(pOrigin,209.5,17.6,0.0),vDraw,z1,tPen\WObj:=wPaper;
    MoveL Offs(pOrigin,211.0,20.5,0.0),vDraw,z1,tPen\WObj:=wPaper;
    MoveL Offs(pOrigin,207.3,30.1,0.0),vDraw,z1,tPen\WObj:=wPaper;
    MoveL Offs(pOrigin,203.6,31.6,0.0),vDraw,z1,tPen\WObj:=wPaper;
    MoveL Offs(pOrigin,200.7,28.7,0.0),vDraw,z1,tPen\WObj:=wPaper;
    MoveL Offs(pOrigin,197.7,18.3,0.0),vDraw,fine,tPen\WObj:=wPaper;
    MoveL Offs(pOrigin,197.7,18.3,15.0),vApproach,z5,tPen\WObj:=wPaper;
    MoveL Offs(pOrigin,225.8,127.0,15.0),vTravel,z5,tPen\WObj:=wPaper;
    MoveL Offs(pOrigin,225.8,127.0,0.0),vApproach,fine,tPen\WObj:=wPaper;
    MoveL Offs(pOrigin,226.5,135.9,0.0),vDraw,z1,tPen\WObj:=wPaper;
    MoveL Offs(pOrigin,219.9,156.6,0.0),vDraw,z1,tPen\WObj:=wPaper;
    MoveL Offs(pOrigin,215.4,155.8,0.0),vDraw,z1,tPen\WObj:=wPaper;
    MoveL Offs(pOrigin,214.7,150.7,0.0),vDraw,z1,tPen\WObj:=wPaper;
    MoveL Offs(pOrigin,219.1,140.3,0.0),vDraw,z1,tPen\WObj:=wPaper;
    MoveL Offs(pOrigin,220.6,128.5,0.0),vDraw,z1,tPen\WObj:=wPaper;
    MoveL Offs(pOrigin,225.8,127.0,0.0),vDraw,fine,tPen\WObj:=wPaper;
    MoveL Offs(pOrigin,225.8,127.0,15.0),vApproach,z5,tPen\WObj:=wPaper;
    MoveL Offs(pOrigin,223.6,128.5,15.0),vTravel,z5,tPen\WObj:=wPaper;
    MoveL Offs(pOrigin,223.6,128.5,0.0),vApproach,fine,tPen\WObj:=wPaper;
    MoveL Offs(pOrigin,216.2,152.9,0.0),vDraw,z1,tPen\WObj:=wPaper;
    MoveL Offs(pOrigin,217.7,154.4,0.0),vDraw,z1,tPen\WObj:=wPaper;
    MoveL Offs(pOrigin,223.6,141.8,0.0),vDraw,z1,tPen\WObj:=wPaper;
    MoveL Offs(pOrigin,225.1,134.4,0.0),vDraw,z1,tPen\WObj:=wPaper;
    MoveL Offs(pOrigin,223.6,128.5,0.0),vDraw,fine,tPen\WObj:=wPaper;
    MoveL Offs(pOrigin,223.6,128.5,15.0),vApproach,z5,tPen\WObj:=wPaper;
    MoveL Offs(pOrigin,195.5,164.7,15.0),vTravel,z5,tPen\WObj:=wPaper;
    MoveL Offs(pOrigin,195.5,164.7,0.0),vApproach,fine,tPen\WObj:=wPaper;
    MoveL Offs(pOrigin,193.3,164.7,0.0),vDraw,z1,tPen\WObj:=wPaper;
    MoveL Offs(pOrigin,188.8,169.2,0.0),vDraw,z1,tPen\WObj:=wPaper;
    MoveL Offs(pOrigin,189.6,174.3,0.0),vDraw,z1,tPen\WObj:=wPaper;
    MoveL Offs(pOrigin,193.3,177.3,0.0),vDraw,z1,tPen\WObj:=wPaper;
    MoveL Offs(pOrigin,198.4,175.8,0.0),vDraw,z1,tPen\WObj:=wPaper;
    MoveL Offs(pOrigin,201.4,171.4,0.0),vDraw,z1,tPen\WObj:=wPaper;
    MoveL Offs(pOrigin,195.5,164.7,0.0),vDraw,fine,tPen\WObj:=wPaper;
    MoveL Offs(pOrigin,195.5,164.7,15.0),vApproach,z5,tPen\WObj:=wPaper;
    MoveL Offs(pOrigin,182.2,158.8,15.0),vTravel,z5,tPen\WObj:=wPaper;
    MoveL Offs(pOrigin,182.2,158.8,0.0),vApproach,fine,tPen\WObj:=wPaper;
    MoveL Offs(pOrigin,180.7,168.4,0.0),vDraw,z1,tPen\WObj:=wPaper;
    MoveL Offs(pOrigin,178.5,169.9,0.0),vDraw,z1,tPen\WObj:=wPaper;
    MoveL Offs(pOrigin,169.6,169.2,0.0),vDraw,z1,tPen\WObj:=wPaper;
    MoveL Offs(pOrigin,166.6,164.0,0.0),vDraw,z1,tPen\WObj:=wPaper;
    MoveL Offs(pOrigin,167.4,157.3,0.0),vDraw,z1,tPen\WObj:=wPaper;
    MoveL Offs(pOrigin,172.6,154.4,0.0),vDraw,z1,tPen\WObj:=wPaper;
    MoveL Offs(pOrigin,179.9,155.8,0.0),vDraw,z1,tPen\WObj:=wPaper;
    MoveL Offs(pOrigin,182.2,158.8,0.0),vDraw,fine,tPen\WObj:=wPaper;
    MoveL Offs(pOrigin,182.2,158.8,15.0),vApproach,z5,tPen\WObj:=wPaper;
    MoveL Offs(pOrigin,179.2,158.8,15.0),vTravel,z5,tPen\WObj:=wPaper;
    MoveL Offs(pOrigin,179.2,158.8,0.0),vApproach,fine,tPen\WObj:=wPaper;
    MoveL Offs(pOrigin,174.8,155.8,0.0),vDraw,z1,tPen\WObj:=wPaper;
    MoveL Offs(pOrigin,168.1,161.0,0.0),vDraw,z1,tPen\WObj:=wPaper;
    MoveL Offs(pOrigin,168.9,164.7,0.0),vDraw,z1,tPen\WObj:=wPaper;
    MoveL Offs(pOrigin,173.3,168.4,0.0),vDraw,z1,tPen\WObj:=wPaper;
    MoveL Offs(pOrigin,177.7,167.7,0.0),vDraw,z1,tPen\WObj:=wPaper;
    MoveL Offs(pOrigin,180.7,164.0,0.0),vDraw,z1,tPen\WObj:=wPaper;
    MoveL Offs(pOrigin,179.2,158.8,0.0),vDraw,fine,tPen\WObj:=wPaper;
    MoveL Offs(pOrigin,179.2,158.8,15.0),vApproach,z5,tPen\WObj:=wPaper;
    MoveL Offs(pOrigin,182.2,175.8,15.0),vTravel,z5,tPen\WObj:=wPaper;
    MoveL Offs(pOrigin,182.2,175.8,0.0),vApproach,fine,tPen\WObj:=wPaper;
    MoveL Offs(pOrigin,177.7,176.5,0.0),vDraw,z1,tPen\WObj:=wPaper;
    MoveL Offs(pOrigin,174.8,180.2,0.0),vDraw,z1,tPen\WObj:=wPaper;
    MoveL Offs(pOrigin,174.8,183.9,0.0),vDraw,z1,tPen\WObj:=wPaper;
    MoveL Offs(pOrigin,179.2,188.4,0.0),vDraw,z1,tPen\WObj:=wPaper;
    MoveL Offs(pOrigin,182.9,188.4,0.0),vDraw,z1,tPen\WObj:=wPaper;
    MoveL Offs(pOrigin,187.3,183.9,0.0),vDraw,z1,tPen\WObj:=wPaper;
    MoveL Offs(pOrigin,186.6,179.5,0.0),vDraw,z1,tPen\WObj:=wPaper;
    MoveL Offs(pOrigin,182.2,175.8,0.0),vDraw,fine,tPen\WObj:=wPaper;
    MoveL Offs(pOrigin,182.2,175.8,15.0),vApproach,z5,tPen\WObj:=wPaper;
  ENDPROC

ENDMODULE
